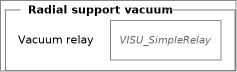
VISUALIZATION VISU_M1RadialSupportVacuum  // 237x72
VAR_IN_OUT
	ref : M1RadialSupport;
    widget : M1RadialSupportWidget;
END_VAR
    Label (15,25 90x30), "Vacuum relay"
    Label (25,0 150x20), "Radial support vacuum"
    Frame (110,20 111x40)
        shows VISU_SimpleRelay(ref := ref.parts.vacuumRelay, widget := widget.vacuumRelay)
    Polyline (20,10) (5,10) (5,70) (235,70) (235,10) (165,10)
END_VISUALIZATION

(* stored: Version 1.1.0.1, ProductVersion 3.1.4019.2
   Visu VISU_M1RadialSupportVacuum: Id {a42a294d-1f2d-4436-8450-4ba4ead26806} *)
